FUNCTION_BLOCK LevelController (* Composite Function Block Type *)
  (* Standard: 61499-2 *)
  (* Version 0.0, 2011-12-18, 4DIAC-IDE, 4DIAC-Consortium *)
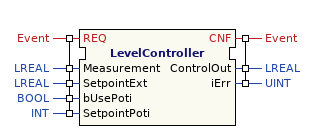
  EVENT_INPUT
    REQ WITH Measurement, SetpointExt, bUsePoti, SetpointPoti; (* Normal Execution Request *)
  END_EVENT
  EVENT_OUTPUT
    CNF WITH ControlOut, iErr; (* Execution Confirmation *)
  END_EVENT
  VAR_INPUT
    Measurement : LREAL; (* Input event qualifier *)
    SetpointExt : LREAL;
    bUsePoti : BOOL;
    SetpointPoti : INT;
  END_VAR
  VAR_OUTPUT
    ControlOut : LREAL; (* Output event qualifier *)
    iErr : UINT;
  END_VAR
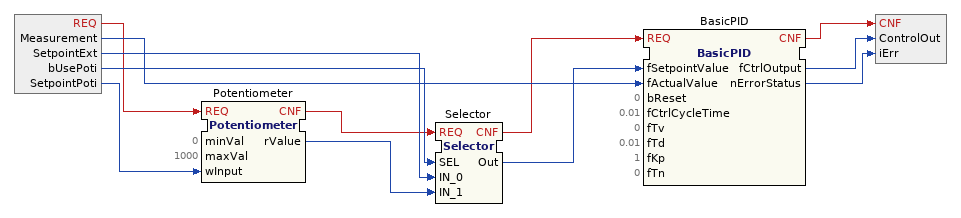
  FBS
    BasicPID : BasicPID(bReset := 0, fCtrlCycleTime := 0.01, fTv := 0, fTd := 0.01, fKp := 1, fTn := 0);
    Potentiometer : Potentiometer(minVal := 0, maxVal := 1000);
    Selector : Selector;
  END_FBS
  EVENT_CONNECTIONS
    BasicPID.CNF TO CNF;
    REQ TO Potentiometer.REQ;
    Selector.CNF TO BasicPID.REQ;
    Potentiometer.CNF TO Selector.REQ;
  END_CONNECTIONS
  DATA_CONNECTIONS
    Measurement TO BasicPID.fActualValue;
    BasicPID.fCtrlOutput TO ControlOut;
    BasicPID.nErrorStatus TO iErr;
    SetpointPoti TO Potentiometer.wInput;
    Selector.Out TO BasicPID.fSetpointValue;
    bUsePoti TO Selector.SEL;
    Potentiometer.rValue TO Selector.IN_1;
    SetpointExt TO Selector.IN_0;
  END_CONNECTIONS
END_FUNCTION_BLOCK
